// TwinCAT 3 PLC project T2Pid_Plc
// Title: T2Pid_Plc
// Company: Tc3 Project
// ProjectVersion: 1.0.0.0
// ProgramVersion: 3.1.4026.22
// libraries:
//   Tc2_Standard, * (Beckhoff Automation GmbH)
//   Tc2_System, * (Beckhoff Automation GmbH)
// project tree:
//   / PlcTask.TcTTO
//   POUs/ FB_Pid.TcPOU, I_Pid.TcIO, MAIN.TcPOU
// real-time tasks:
//   TASK PlcTask: cycle T#10ms, priority 20, ADS port 350

CONFIGURATION T2Pid_Plc
    RESOURCE PLC ON TwinCAT3
        TASK PlcTask(INTERVAL := T#10ms, PRIORITY := 20);
        PROGRAM MAIN WITH PlcTask : MAIN;
    END_RESOURCE
END_CONFIGURATION

// ---- POUs/I_Pid.TcIO
INTERFACE I_Pid

METHOD Reset
END_METHOD

METHOD Update : LREAL
VAR_INPUT
    setpoint    : LREAL;
    measurement : LREAL;
    deltaT      : LREAL;
END_VAR
END_METHOD

END_INTERFACE

// ---- POUs/MAIN.TcPOU
PROGRAM MAIN
VAR
END_VAR

END_PROGRAM

// ---- POUs/FB_Pid.TcPOU
FUNCTION_BLOCK FB_Pid
VAR
END_VAR

END_FUNCTION_BLOCK
